(* PLC project Unnamed, Unknown Unnamed 1 *)
(* stored: creationDateTime 2025-09-08T14:55:38, modificationDateTime 2025-09-09T14:11:03 *)

PROGRAM Conveyor
  VAR_INPUT
    START_BTN : BOOL;
    STOP_BTN : BOOL;
    S_LARGE : BOOL;
    E_STOP : BOOL;
  END_VAR
  VAR_OUTPUT
    M_CONV : BOOL;
    DIVERT : BOOL;
  END_VAR
  VAR
    RUN_CMD AT %MX0.0 : BOOL;
    RUN_CMD0 AT %MX0.1 : BOOL;
  END_VAR
  VAR
    TP0 : TP;
  END_VAR
  VAR_INPUT
    SORT_TIME : TIME := T#3s;
  END_VAR

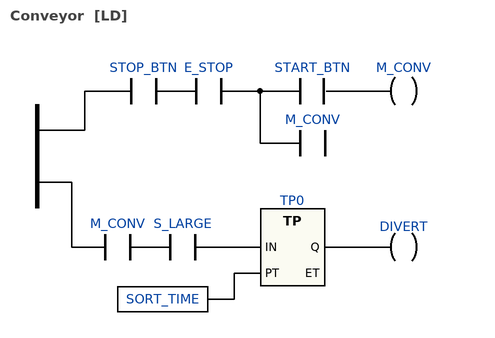
(* LD diagram, written out as Structured Text *)
M_CONV := STOP_BTN AND E_STOP AND START_BTN;
TP0(IN := M_CONV AND S_LARGE, PT := SORT_TIME);
DIVERT := TP0.Q;
(* drawn but not wired to any output: M_CONV *)
END_PROGRAM

CONFIGURATION Config0
  RESOURCE Res0 ON PLC
    TASK task0(INTERVAL := T#20ms, PRIORITY := 0);
    PROGRAM instance0 WITH task0 : Conveyor;
  END_RESOURCE
END_CONFIGURATION
